// TIA Portal V20 export
ORGANIZATION_BLOCK "Main"   // OB1, LAD, ProgramCycle
TITLE = "Main Program Sweep (Cycle)"
// stored: IsIECCheckEnabled true, SetENOAutomatically false
   VAR_INPUT
      Initial_Call : Bool;   // Initial call of this OB
      Remanence : Bool;   // =True, if remanent data are available
   END_VAR
BEGIN

REGION Network 1: New comment
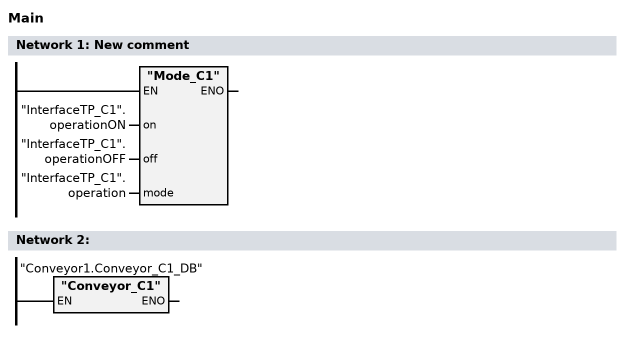
   RUNG wire#powerrail
      "Mode_C1"(on := "InterfaceTP_C1".operationON, off := "InterfaceTP_C1".operationOFF, mode := "InterfaceTP_C1".operation)
   END_RUNG
   // the same network as SCL:
   "Mode_C1"(on := "InterfaceTP_C1".operationON,
             off := "InterfaceTP_C1".operationOFF,
             mode := "InterfaceTP_C1".operation);
END_REGION

REGION Network 2
   RUNG wire#powerrail
      "Conveyor1.Conveyor_C1_DB"()
   END_RUNG
   // the same network as SCL:
   "Conveyor1.Conveyor_C1_DB"();   // "Conveyor_C1"
END_REGION
END_ORGANIZATION_BLOCK
